{attribute 'GeneratedUsingTerminal: EK1122-0000-0018'}
{attribute addProperty BoxType "EK1122-0000-0018"}
{attribute addProperty Id "Beckhoff_EKx9xxsub_EK1100EK1100_AB5A94672A_0001_EK1960_0000_0019EK1960_B44B3219142A_0002_EK1960_0000_0021EK1960_3972CFDA138A_0003_EK1960_0008_0019EK1960_B44B3219142A_0004_EK1960_0008_0021EK1960_3972CFDA138A_0005_EK1960_2600_0019EK1960_39B343E2148A_0006_EK1960_2600_0021EK1960_A744D3A0148A_0007_EK1960_2608_0019EK1960_39B343E2148A_0008_EK1960_2608_0021EK1960_A744D3A0148"}
{attribute addProperty CRC "1133686048"}
{attribute addProperty Size "1154"}
TYPE Beckhoff_EKx9xxEK1122_4392AD20 EXTENDS EK1122_AB5A9467 :
STRUCT
	{attribute addProperty Name "Beckhoff_EKx9xxsub_EK1100"}
	{attribute addProperty PreviousPort "Beckhoff EKx9xxEK1122 : D"}
	Beckhoff_EKx9xxsub_EK1100 : EK1100_AB5A9467;
	{attribute addProperty Name "A_0001_EK1960_0000_0019"}
	{attribute addProperty PreviousPort "Beckhoff EKx9xxsub EK1100 : C"}
	A_0001_EK1960_0000_0019 : EK1960_B44B3219;
	{attribute addProperty Name "A_0002_EK1960_0000_0021"}
	{attribute addProperty PreviousPort "A_0001(EK1960-0000-0019) : C"}
	A_0002_EK1960_0000_0021 : EK1960_3972CFDA;
	{attribute addProperty Name "A_0003_EK1960_0008_0019"}
	{attribute addProperty PreviousPort "A_0002(EK1960-0000-0021) : C"}
	A_0003_EK1960_0008_0019 : EK1960_B44B3219;
	{attribute addProperty Name "A_0004_EK1960_0008_0021"}
	{attribute addProperty PreviousPort "A_0003(EK1960-0008-0019) : C"}
	A_0004_EK1960_0008_0021 : EK1960_3972CFDA;
	{attribute addProperty Name "A_0005_EK1960_2600_0019"}
	{attribute addProperty PreviousPort "A_0004(EK1960-0008-0021) : C"}
	A_0005_EK1960_2600_0019 : EK1960_39B343E2;
	{attribute addProperty Name "A_0006_EK1960_2600_0021"}
	{attribute addProperty PreviousPort "A_0005(EK1960-2600-0019) : C"}
	A_0006_EK1960_2600_0021 : EK1960_A744D3A0;
	{attribute addProperty Name "A_0007_EK1960_2608_0019"}
	{attribute addProperty PreviousPort "A_0006(EK1960-2600-0021) : C"}
	A_0007_EK1960_2608_0019 : EK1960_39B343E2;
	{attribute addProperty Name "A_0008_EK1960_2608_0021"}
	{attribute addProperty PreviousPort "A_0007(EK1960-2608-0019) : C"}
	A_0008_EK1960_2608_0021 : EK1960_A744D3A0;
END_STRUCT
END_TYPE

(* stored: Version 1.2.0.0, ProductVersion 3.1.4024.9
   DUT Beckhoff_EKx9xxEK1122_4392AD20: Id {c9688551-3f69-4c22-b6c8-64ed0cce0479} *)
